{attribute 'qualified_only'}
VAR_GLOBAL
	ActualStep : BYTE := 1;
END_VAR

(* stored: Version 1.1.0.1, ProductVersion 3.1.4024.13
   GVL Steps: Id {fdf35bbd-ce64-48d9-9622-ce868d6165e0} *)
